FUNCTION DHTrans : ST_Frame
VAR_IN_OUT CONSTANT
	// DH parameters: alpha, a, d, DH[4]
	DH :Vec4d;
END_VAR
VAR
END_VAR

DHTrans.m_rot[1,1]:= COS(DH[4]);
DHTrans.m_rot[1,2]:=  -SIN(DH[4]);
DHTrans.m_rot[1,3]:= 0;
DHTrans.m_rot[2,1]:= COS(DH[1])*SIN(DH[4]);
DHTrans.m_rot[2,2]:= COS(DH[1])*COS(DH[4]);
DHTrans.m_rot[2,3]:= -SIN(DH[1]);
DHTrans.m_rot[3,1]:= SIN(DH[1])*SIN(DH[4]);
DHTrans.m_rot[3,2]:= SIN(DH[1])*COS(DH[4]);
DHTrans.m_rot[3,3]:= COS(DH[1]);

DHTrans.m_pos[1]:=DH[2];
DHTrans.m_pos[2]:=-DH[3]*SIN(DH[1]);
DHTrans.m_pos[3]:=DH[3]*COS(DH[1]);

END_FUNCTION

(* stored: Version 1.1.0.1, ProductVersion 3.1.4024.12
   POU DHTrans: Id {6f2f5444-d30f-44ea-b23b-d19608633eba}, SpecialFunc None *)
